Staubli VAL3: create.pgx

public program create(num x_nDetNum, string x_sTask)
begin
  call init(x_nDetNum,x_sTask)
  taskCreate sTASK,100,detection()
end
